FUNCTION_BLOCK DigitalInput (* CAT Function Block Type *)
  (* Standard: 61499-2 *)
  (* Version 0.0, 6/15/2026, Schneider Electric, template *)
  PACKAGE SE.Nereda;
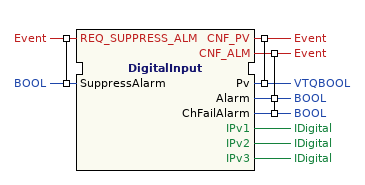
  EVENT_INPUT
    REQ_SUPPRESS_ALM WITH SuppressAlarm; (* Request to suppress alarms *)
  END_EVENT
  EVENT_OUTPUT
    CNF_PV WITH Pv; (* Execution confirmation of Pv *)
    CNF_ALM WITH Alarm, ChFailAlarm; (* Execution confirmation of alarm *)
  END_EVENT
  VAR_INPUT
    SuppressAlarm : BOOL; (* 1 = Suppress channel failure and state alarm monitoring in HMI *)
  END_VAR
  VAR_OUTPUT
    Pv : VTQBOOL; (* Process value output *)
    Alarm : BOOL; (* 1 = State alarm is active *)
    ChFailAlarm : BOOL; (* 1 = Alarm is active *)
  END_VAR
  PLUGS
    IPv1 : IDigital; (* Process value interface adapter *)
    IPv2 : IDigital; (* Process value interface adapter *)
    IPv3 : IDigital; (* Process value interface adapter *)
  END_PLUGS
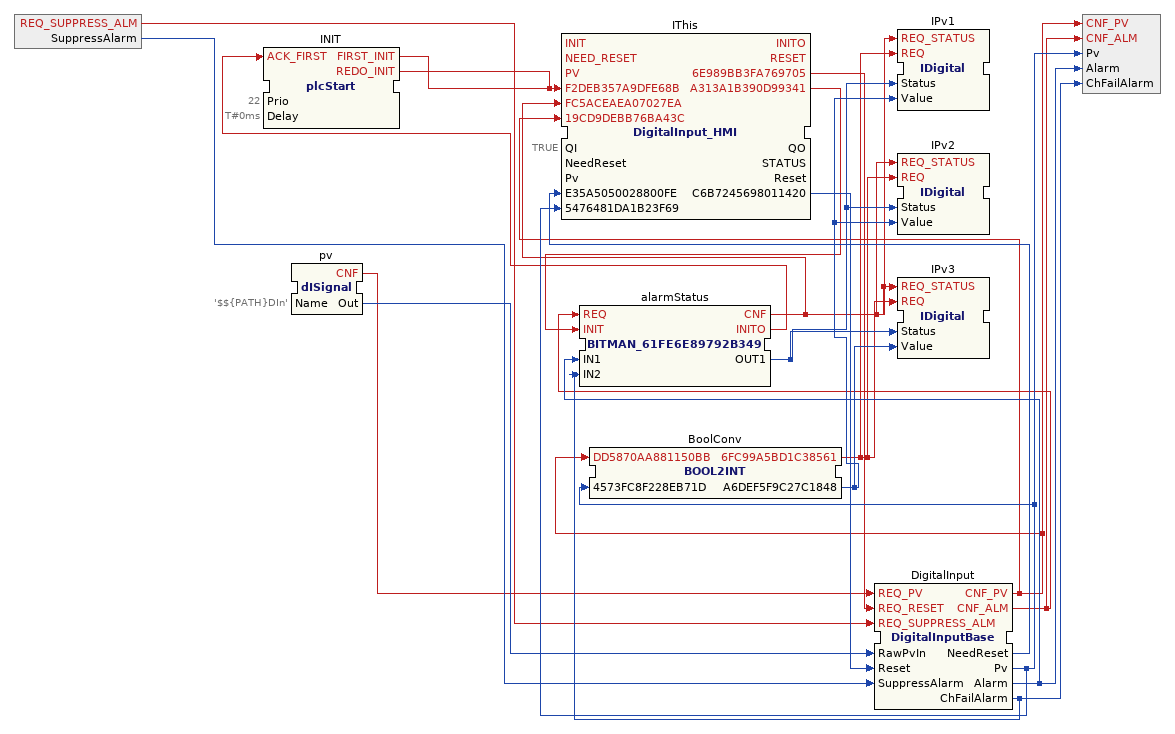
  (* 01 - FUNCTIONNAL INPUT INTERFACE *)
  (* 00 - INITIALIZATION *)
  (* 05 - LOGIC *)
  (* 06 - HMI INTERFACE *)
  (* 04 - CHILDREN *)
  (* 03 - FIELD INTERFACE *)
  (* 02 - FUNCTIONNAL OUTPUT INTERFACE *)
  (* 07- Input Hardware Interface *)
  (* 4A - TYPICALS *)
  (* Alarm Status *)
  FBS
    INIT : plcStart(Prio := 22, Delay := T#0ms);
    IThis : DigitalInput_HMI(QI := TRUE);
    DigitalInput : DigitalInputBase;
    pv : dISignal(Name := '$${PATH}DIn');
    alarmStatus : BITMAN_61FE6E89792B349; {SET_ATTRIBUTE(Configuration.GenericFBType.InterfaceParams, Runtime.Standard#CNTIN:=2;CNTOUT:=1;IN${CNTIN$}:BOOL,BOOL;OUT${CNTOUT$}:WORD)}
    BoolConv : BOOL2INT;
  END_FBS
  EVENT_CONNECTIONS
    pv.CNF TO DigitalInput.REQ_PV;
    alarmStatus.CNF TO IPv1.REQ_STATUS;
    INIT.FIRST_INIT TO IThis.F2DEB357A9DFE68B;
    INIT.REDO_INIT TO IThis.F2DEB357A9DFE68B;
    alarmStatus.CNF TO IThis.FC5ACEAEA07027EA;
    DigitalInput.CNF_PV TO IThis.19CD9DEBB76BA43C;
    alarmStatus.INITO TO INIT.ACK_FIRST;
    IThis.6E989BB3FA769705 TO DigitalInput.REQ_RESET;
    DigitalInput.CNF_ALM TO alarmStatus.REQ;
    IThis.A313A1B390D99341 TO alarmStatus.INIT;
    REQ_SUPPRESS_ALM TO DigitalInput.REQ_SUPPRESS_ALM;
    DigitalInput.CNF_PV TO CNF_PV;
    DigitalInput.CNF_ALM TO CNF_ALM;
    alarmStatus.CNF TO IPv2.REQ_STATUS;
    alarmStatus.CNF TO IPv3.REQ_STATUS;
    DigitalInput.CNF_PV TO BoolConv.DD5870AA881150BB;
    BoolConv.6FC99A5BD1C38561 TO IPv1.REQ;
    BoolConv.6FC99A5BD1C38561 TO IPv2.REQ;
    BoolConv.6FC99A5BD1C38561 TO IPv3.REQ;
  END_CONNECTIONS
  DATA_CONNECTIONS
    pv.Out TO DigitalInput.RawPvIn;
    DigitalInput.NeedReset TO IThis.E35A5050028800FE;
    DigitalInput.Pv TO IThis.5476481DA1B23F69;
    IThis.C6B7245698011420 TO DigitalInput.Reset;
    alarmStatus.OUT1 TO IPv1.Status;
    DigitalInput.Alarm TO alarmStatus.IN1;
    DigitalInput.ChFailAlarm TO alarmStatus.IN2;
    SuppressAlarm TO DigitalInput.SuppressAlarm;
    DigitalInput.Pv TO Pv;
    DigitalInput.Alarm TO Alarm;
    DigitalInput.ChFailAlarm TO ChFailAlarm;
    alarmStatus.OUT1 TO IPv2.Status;
    alarmStatus.OUT1 TO IPv3.Status;
    DigitalInput.Pv TO BoolConv.4573FC8F228EB71D;
    BoolConv.A6DEF5F9C27C1848 TO IPv1.Value;
    BoolConv.A6DEF5F9C27C1848 TO IPv2.Value;
    BoolConv.A6DEF5F9C27C1848 TO IPv3.Value;
  END_CONNECTIONS
END_FUNCTION_BLOCK
